VAR_GLOBAL CONSTANT
	
	gNUM_MOVERS		: USINT := 6;
	gNUM_STATIONS	: USINT := 4;

END_VAR

(* stored: Version 1.1.0.1, ProductVersion 3.1.4024.9
   GVL XTS_Constants: Id {243a1f03-dc04-4ddf-a082-a0f0db6d0ff8}, ParameterList True *)
